// TIA Portal V19 export
TYPE "C205_VAR_IF_GVL_TYPIC"
   STRUCT
      BMO_AAN { ExternalAccessible := 'False'; ExternalVisible := 'False'; ExternalWritable := 'False'} : Bool;   // Geleideverlichting aan
      EXT_AUT { ExternalAccessible := 'False'; ExternalVisible := 'False'; ExternalWritable := 'False'} : Bool;   // Externe (hoofd) beveiliging aangesproken
      EXT_HW { ExternalAccessible := 'False'; ExternalVisible := 'False'; ExternalWritable := 'False'} : Bool;   // Sturings hardware (PLC) in storing
      STO { ExternalAccessible := 'False'; ExternalVisible := 'False'; ExternalWritable := 'False'} : Struct   // Opsomming van alle storingen en meldingen
         A001 : Bool;   // Beveiliging aangesproken
         A002 : Bool;   // Storing voeding geleideverlichting
         AT01 : Bool;   // Foute terugmelding: Geleideverlichting aangestuurd, terugmelding Aan niet (of te laat) ontvangen
         AT02 : Bool;   // Foute terugmelding: Geleideverlichting niet aangestuurd, terugmelding Aan blijft aanwezig
      END_STRUCT;
   END_STRUCT;
END_TYPE
